FUNCTION_BLOCK Motor IMPLEMENTS itfAutoManual
VAR_INPUT
	MotorInput : MotorI;
END_VAR
VAR_OUTPUT
	MotorOutput : MotorO;
END_VAR
VAR
	Actuate : itfActuate;
	Fault : itfFault;
	
	ActuateComp : itfActuateImplement;
	FaultComp : itfFaultImplement;
END_VAR

Map();
FaultHandler();

METHOD PROTECTED FaultHandler : BOOL
VAR_INPUT
END_VAR
Fault.mResetFault();
Fault.mSetFault();
END_METHOD

METHOD PRIVATE Map : BOOL
VAR_INPUT
END_VAR
Actuate := ActuateComp;
Fault := FaultComp;

Actuate.pStart := MotorInput.Start;
Actuate.pStop := MotorInput.Stop;
MotorOutput.Coil := Actuate.pCoil;
MotorOutput.FaultStatus := Fault.pFaultStatus;

Fault.pResetButton := MotorInput.ResetOverload;
Fault.pFault := MotorInput.Overload;
END_METHOD

{warning 'add method implementation '}
METHOD mAutoOff : BOOL
Actuate.mTurnOffAuto();
END_METHOD

{warning 'add method implementation '}
METHOD mAutoOn : BOOL
IF mFault() = FALSE THEN
Actuate.mTurnOnAuto();
END_IF
END_METHOD

{warning 'add method implementation '}
METHOD mFault : BOOL
mFault := Fault.pFaultStatus;
END_METHOD

{warning 'add method implementation '}
METHOD mManual : BOOL
IF mFault() = FALSE THEN
Actuate.mTurnOnManual();
END_IF
Actuate.mTurnOffManual();
END_METHOD

{warning 'add method implementation '}
METHOD mRunning : BOOL
mRunning := Actuate.pCoil;
END_METHOD

END_FUNCTION_BLOCK

(* stored: Version 1.1.0.1, ProductVersion 3.1.4024.12
   POU Motor: Id {3cbfe4dd-9e30-4896-a5f5-8ef056504abb}, SpecialFunc None
   Method FaultHandler: Id {f393ba9e-00a6-4f68-aa72-1db891210240}
   Method Map: Id {86d08d12-b511-4f03-a9cb-b78cff376b33}
   Method mAutoOff: Id {4d3edd47-c467-48f4-8a9f-cee0adb9c444}
   Method mAutoOn: Id {ebfc1c94-d6b8-4a45-9091-987d607a6613}
   Method mFault: Id {5a3c9ec4-5a53-42ac-9e00-7832b09da4d8}
   Method mManual: Id {9c5b2efa-38a4-4abd-88a7-77a9dc2fa2e1}
   Method mRunning: Id {b523a23e-6d71-4392-8359-8585efa9b969} *)
